(* PLC project tni_clock, Dassault Systèmes ControlBuild 2024x *)
(* stored: creationDateTime 2023-10-03T11:13:48-01:00 *)

PROGRAM tni_clock.tni_clock
  VAR_IN_OUT
    B1 : BOOL := false;
    B2 : BOOL := false;
    B3 : BOOL := false;
    B4 : BOOL := false;
  END_VAR
  VAR_INPUT
    depth : INT := 0;
  END_VAR

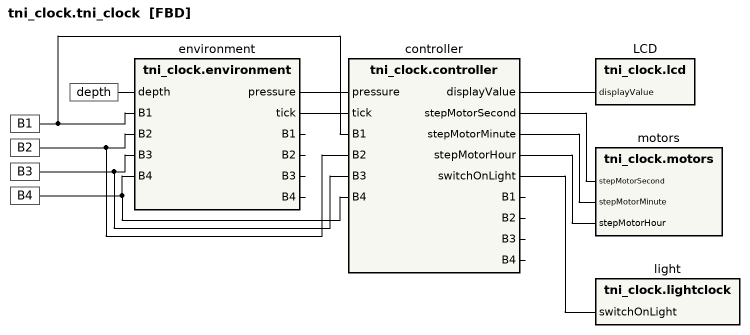
(* FBD diagram, written out as Structured Text *)
environment(depth := depth, B1 := B1, B2 := B2, B3 := B3, B4 := B4);
controller(pressure := environment.pressure, tick := environment.tick, B1 := B1, B2 := B2, B3 := B3, B4 := B4);
LCD(displayValue := controller.displayValue);
motors(stepMotorSecond := controller.stepMotorSecond, stepMotorMinute := controller.stepMotorMinute, stepMotorHour := controller.stepMotorHour);
light(switchOnLight := controller.switchOnLight);
END_PROGRAM
